FUNCTION_BLOCK EL3054
VAR
	_io : EL3xx4_Data;
	{attribute addProperty Name "WcState"}
	_wcState : WcStateInputToggle;
	{attribute addProperty Name "Info data"}
	_infoData : InfoDataAds;
END_VAR

PROPERTY IO : REFERENCE TO EL3xx4_Data
GET
IO REF= _io;
END_GET
END_PROPERTY

PROPERTY WcState : REFERENCE TO WcStateInputToggle
GET
WcState REF= _wcState;
END_GET
END_PROPERTY

END_FUNCTION_BLOCK

(* stored: Version 1.1.0.1, ProductVersion 3.1.4024.9
   POU EL3054: Id {ce8c10ee-857d-0b31-00d0-b811f9ff540d}, SpecialFunc None
   Property IO: Id {0331b8ec-9b0c-0f6f-310b-220aca086ba1}
   Get Get: Id {fd9bbfef-6344-0cc0-07ea-de941af58c77}
   Property WcState: Id {0ded793c-3792-07c9-0b81-20f8f855952d}
   Get Get: Id {0ca8ae4c-d447-0171-3ed1-231d669f551f} *)
